// Retrieves information about the target.
{attribute 'no_explicit_call' := 'direct call for this program is not allowed'} 
PROGRAM P_GetSystemInformation

// The version as defined in the compile options.
PROPERTY CompilerVersion : VERSION
GET
CompilerVersion := __SYSTEM.Constants.CompilerVersion;
END_GET
END_PROPERTY

// The version as defined in the compile options.
PROPERTY CompilerVersionNumeric : DWORD
GET
CompilerVersionNumeric := __SYSTEM.Constants.CompilerVersionNumeric;
END_GET
END_PROPERTY

// Indicates of whether the target has FPU support.
PROPERTY HasFpuSupport : BOOL
GET
HasFpuSupport := __SYSTEM.Constants.bFPUSupport;
END_GET
END_PROPERTY

// Indicates whether multicore support is available in the target.
PROPERTY HasMulticoreSupport : BOOL
GET
HasMulticoreSupport := __SYSTEM.Constants.bMulticoreSupport;
END_GET
END_PROPERTY

// Indicates if target is in simulation mode.
PROPERTY InSimulationMode : BOOL
GET
InSimulationMode := __SYSTEM.Constants.bSimulationMode;
END_GET
END_PROPERTY

// Indicates of the system is little endian; TRUE for Intel, ARM etc. FALSE for Power PC, etc. 
PROPERTY IsLittleEndian : BOOL
GET
IsLittleEndian := __SYSTEM.Constants.bLittleEndian;
END_GET
END_PROPERTY

// Retrieves the operating system of the target.
PROPERTY OperatingSystem : E_OperatingSystem
GET
VAR_STAT
	nOperatingSystem : UDINT;
	nResult : UDINT := SysTarget.SysTargetGetOperatingSystemId(ADR(nOperatingSystem));
END_VAR
CASE nOperatingSystem OF
	1..4: OperatingSystem := E_OperatingSystem.Windows;
	5: OperatingSystem := E_OperatingSystem.Linux;
	6: OperatingSystem := E_OperatingSystem.VxWorks;
	7: OperatingSystem := E_OperatingSystem.QNX;
	8: OperatingSystem := E_OperatingSystem.uCOS;
ELSE
	OperatingSystem := E_OperatingSystem._;
	END_CASE
END_GET
END_PROPERTY

// Retrieves the packmode of the system.
PROPERTY PackMode : WORD
GET
PackMode := __SYSTEM.Constants.nPackMode;
END_GET
END_PROPERTY

// Retireves the target's processor architecture.
PROPERTY ProcessorArchitecture : E_ProcessorArchitecture
GET
VAR_STAT
	nProcessorArchitecture : UDINT;
	nResult : UDINT := SysTarget.SysTargetGetProcessorId(ADR(nProcessorArchitecture));
END_VAR
ProcessorArchitecture := TO_BYTE(nProcessorArchitecture);
END_GET
END_PROPERTY

// Retrieves the size of the CPU register; 16 for C16x, 64 for X86-64 Bit, 32 for all other controllers.
PROPERTY RegisterSize : WORD
GET
RegisterSize := __SYSTEM.Constants.nRegisterSize;
END_GET
END_PROPERTY

// The version as described in the runtime system.
PROPERTY RuntimeVersion : VERSION
GET
RuntimeVersion := __SYSTEM.Constants.RuntimeVersion;
END_GET
END_PROPERTY

// The version as described in the runtime system.
PROPERTY RuntimeVersionNumeric : DWORD
GET
RuntimeVersionNumeric := __SYSTEM.Constants.RuntimeVersionNumeric;
END_GET
END_PROPERTY

END_PROGRAM

(* stored: Version 1.1.0.1
   POU P_GetSystemInformation: Id {b0e883b6-90aa-0c6d-36b2-0947b0933caf}, SpecialFunc None
   Property CompilerVersion: Id {91c1a12c-b37a-0e19-3119-cb82109908df}
   Get Get: Id {cf466b9a-2f5e-03e0-2ba5-607787a2daac}
   Property CompilerVersionNumeric: Id {e7e5d7f4-c05a-0402-0984-b83bedbdc6b1}
   Get Get: Id {3cd18d96-b606-0fe6-05b0-8a3efb458b26}
   Property HasFpuSupport: Id {32b283c3-d4ba-0270-0f42-5b7e5edc3922}
   Get Get: Id {626ccf4d-7625-0b2b-0ce6-7a56bb32ff7d}
   Property HasMulticoreSupport: Id {4df5d3ab-89dc-060c-1bb9-c38dfe82a90d}
   Get Get: Id {4e423ab2-d2fe-0d5d-2003-ddc7f2102e08}
   Property InSimulationMode: Id {5ab8d195-09ee-05f2-36e4-d250a2eb8bf4}
   Get Get: Id {4615fa1d-230f-06da-0386-bacf0b1b2a30}
   Property IsLittleEndian: Id {a7992363-dceb-0a16-287d-0f34eee98d47}
   Get Get: Id {a14cc85e-b4af-0024-156a-543f1181f1dc}
   Property OperatingSystem: Id {336cc389-1120-079a-326a-175db3d2f3fb}
   Get Get: Id {6ab1df7c-3a9b-0280-106b-51fc293e59e6}
   Property PackMode: Id {7452dbaa-8d53-0e32-1ccc-970af7901e03}
   Get Get: Id {a98370b3-63d6-0bef-2306-0ebcf32cb17f}
   Property ProcessorArchitecture: Id {6b336d92-e78b-0b30-0721-8bc6141fb57c}
   Get Get: Id {520417e0-26ec-0961-2c1d-de4d1180fee7}
   Property RegisterSize: Id {47268eef-7ba3-092f-1329-da4031e647cb}
   Get Get: Id {740e8e51-6ff8-02e9-0958-e23b0ccf06e1}
   Property RuntimeVersion: Id {584e5609-0718-0ae7-2267-f4de2db2f208}
   Get Get: Id {cde43abf-fc36-0904-312a-05e1680c8f37}
   Property RuntimeVersionNumeric: Id {5a19fa5d-847c-03b5-111a-dde1054fed86}
   Get Get: Id {fa713d99-3d31-04b3-3c56-4e1953f1d2c9} *)
